// TwinCAT 3 PLC project TcLogTest
// ProgramVersion: 3.1.4023.0
// libraries:
//   Tc2_Standard, * (Beckhoff Automation GmbH)
//   Tc2_System, * (Beckhoff Automation GmbH)
//   Tc2_Utilities, * (Beckhoff Automation GmbH)
//   Tc3_Module, * (Beckhoff Automation GmbH)
//   TcLog, * (Benedikt Geisler)
//   TcUnit, * (www.tcunit.org)
// project tree:
//   / MAIN.TcPOU (not stored), PlcTask.TcTTO
//   TwinCAT/ ConvertAnyToString_TEST.TcPOU, DateTime_TEST.TcPOU, DynamicStringBuffer_TEST.TcPOU
//   NET/ TestWrapper_NET.TcPOU
// (motion and I/O tree: see PLC project tclog)
// real-time tasks:
//   TASK PlcTask1: cycle T#10ms, priority 21, ADS port 351

CONFIGURATION TcLogTest
    RESOURCE PLC ON TwinCAT3
        TASK PlcTask(INTERVAL := T#10ms, PRIORITY := 21);
        PROGRAM TESTS WITH PlcTask : TESTS;
    END_RESOURCE
END_CONFIGURATION

// ---- TwinCAT/ConvertAnyToString_TEST.TcPOU
FUNCTION_BLOCK ConvertAnyToString_TEST EXTENDS TcUnit.FB_TestSuite

ConvertAnyByteToString();
ConvertAnyDateAndTimeToString();
ConvertAnyDateToString();
ConvertAnyDINTToString();
ConvertAnyDTToString();
ConvertAnyINTToString();
ConvertAnyLINTToString();
ConvertAnyLRealToString();
ConvertAnyLWordToString();
ConvertAnyRealToString();
ConvertAnySINTToString();
ConvertAnyStringToString();
ConvertAnyTimeToString();
ConvertAnyTODToString();
ConvertAnyUDINTToString();
ConvertAnyUINTToString();
ConvertAnyULINTToString();
ConvertAnyUSINTToString();
ConvertAnyWordToString();
ConvertAnyWStringToString();

METHOD ConvertAnyByteToString : BOOL
VAR
	input : BYTE := 1;
	result : STRING;
	expected : STRING := '1';
END_VAR
TEST('ConvertAnyByteToString');
 
result := AnyToString(input);
 
AssertEquals(Expected := expected,
             Actual := result,
             Message := FormatResult(expected, result));
 
TEST_FINISHED();
END_METHOD

METHOD ConvertAnyDateAndTimeToString : BOOL
VAR
	input : DATE_AND_TIME := DT#1970-01-01-00:00;
	result : STRING;
	expected : STRING := 'DT#1970-01-01-00:00:00';
END_VAR
TEST('ConvertAnyDateAndTimeToString');
 
result := AnyToString(input);
 
AssertEquals(Expected := expected,
             Actual := result,
             Message := FormatResult(expected, result));
 
TEST_FINISHED();
END_METHOD

METHOD ConvertAnyDateToString : BOOL
VAR
	input : DATE := D#1970-01-01;
	result : STRING;
	expected : STRING := 'D#1970-01-01';
END_VAR
TEST('ConvertAnyDateToString');
 
result := AnyToString(input);
 
AssertEquals(Expected := expected,
             Actual := result,
             Message := FormatResult(expected, result));
 
TEST_FINISHED();
END_METHOD

METHOD ConvertAnyDINTToString : BOOL
VAR
	input : DINT := 1;
	result : STRING;
	expected : STRING := '1';
END_VAR
TEST('ConvertAnyDINTToString');
 
result := AnyToString(input);
 
AssertEquals(Expected := expected,
             Actual := result,
             Message := FormatResult(expected, result));
 
TEST_FINISHED();
END_METHOD

METHOD ConvertAnyDTToString : BOOL
VAR
	input : DT := DT#1970-01-01-00:00;
	result : STRING;
	expected : STRING := 'DT#1970-01-01-00:00:00';
END_VAR
TEST('ConvertAnyDTToString');
 
result := AnyToString(input);
 
AssertEquals(Expected := expected,
             Actual := result,
             Message := FormatResult(expected, result));
 
TEST_FINISHED();
END_METHOD

METHOD ConvertAnyDWordToString : BOOL
VAR
	input : DWORD := 1;
	result : STRING;
	expected : STRING := '1';
END_VAR
TEST('ConvertAnyDWordToString');
 
result := AnyToString(input);
 
AssertEquals(Expected := expected,
             Actual := result,
             Message := FormatResult(expected, result));
 
TEST_FINISHED();
END_METHOD

METHOD ConvertAnyINTToString : BOOL
VAR
	input : INT := 1;
	result : STRING;
	expected : STRING := '1';
END_VAR
TEST('ConvertAnyINTToString');
 
result := AnyToString(input);
 
AssertEquals(Expected := expected,
             Actual := result,
             Message := FormatResult(expected, result));
 
TEST_FINISHED();
END_METHOD

METHOD ConvertAnyLINTToString : BOOL
VAR
	input : LINT := 1;
	result : STRING;
	expected : STRING := '1';
END_VAR
TEST('ConvertAnyLINTToString');
 
result := AnyToString(input);
 
AssertEquals(Expected := expected,
             Actual := result,
             Message := FormatResult(expected, result));
 
TEST_FINISHED();
END_METHOD

METHOD ConvertAnyLRealToString : BOOL
VAR
	input : REAL := 1.0;
	result : STRING;
	expected : STRING := '1.0';
END_VAR
TEST('ConvertAnyRealToString');
 
result := AnyToString(input);
 
AssertEquals(Expected := expected,
             Actual := result,
             Message := FormatResult(expected, result));
 
TEST_FINISHED();
END_METHOD

METHOD ConvertAnyLWordToString : BOOL
VAR
	input : LWORD := 1;
	result : STRING;
	expected : STRING := '1';
END_VAR
TEST('ConvertAnyLWordToString');
 
result := AnyToString(input);
 
AssertEquals(Expected := expected,
             Actual := result,
             Message := FormatResult(expected, result));
 
TEST_FINISHED();
END_METHOD

METHOD ConvertAnyRealToString : BOOL
VAR
	input : LREAL := 1.0;
	result : STRING;
	expected : STRING := '1.0';
END_VAR
TEST('ConvertAnyLRealToString');
 
result := AnyToString(input);
 
AssertEquals(Expected := expected,
             Actual := result,
             Message := FormatResult(expected, result));
 
TEST_FINISHED();
END_METHOD

METHOD ConvertAnySINTToString : BOOL
VAR
	input : SINT := 1;
	result : STRING;
	expected : STRING := '1';
END_VAR
TEST('ConvertAnySINTToString');
 
result := AnyToString(input);
 
AssertEquals(Expected := expected,
             Actual := result,
             Message := FormatResult(expected, result));
 
TEST_FINISHED();
END_METHOD

METHOD ConvertAnyStringToString : BOOL
VAR
	input : STRING := 'Hallo';
	result : STRING;
	expected : STRING := 'Hallo';
END_VAR
TEST('ConvertAnyStringToString');
 
result := AnyToString(input);
 
AssertEquals(Expected := expected,
             Actual := result,
             Message := FormatResult(expected, result));
 
TEST_FINISHED();
END_METHOD

METHOD ConvertAnyTimeToString : BOOL
VAR
	input : TIME := T#49D17H2M47S295MS;
	result : STRING;
	expected : STRING := 'T#49d17h2m47s295ms';
END_VAR
TEST('ConvertAnyTimeToString');
 
result := AnyToString(input);
 
AssertEquals(Expected := expected,
             Actual := result,
             Message := FormatResult(expected, result));
 
TEST_FINISHED();
END_METHOD

METHOD ConvertAnyTODToString : BOOL
VAR
	input : TOD := TOD#11:02:47.295;
	result : STRING;
	expected : STRING := 'TOD#11:02:47.295';
END_VAR
TEST('ConvertAnyTODToString');
 
result := AnyToString(input);
 
AssertEquals(Expected := expected,
             Actual := result,
             Message := FormatResult(expected, result));
 
TEST_FINISHED();
END_METHOD

METHOD ConvertAnyUDINTToString : BOOL
VAR
	input : UDINT := 1;
	result : STRING;
	expected : STRING := '1';
END_VAR
TEST('ConvertAnyUDINTToString');
 
result := AnyToString(input);
 
AssertEquals(Expected := expected,
             Actual := result,
             Message := FormatResult(expected, result));
 
TEST_FINISHED();
END_METHOD

METHOD ConvertAnyUINTToString : BOOL
VAR
	input : UINT := 1;
	result : STRING;
	expected : STRING := '1';
END_VAR
TEST('ConvertAnyUINTToString');
 
result := AnyToString(input);
 
AssertEquals(Expected := expected,
             Actual := result,
             Message := FormatResult(expected, result));
 
TEST_FINISHED();
END_METHOD

METHOD ConvertAnyULINTToString : BOOL
VAR
	input : ULINT := 1;
	result : STRING;
	expected : STRING := '1';
END_VAR
TEST('ConvertAnyULINTToString');
 
result := AnyToString(input);
 
AssertEquals(Expected := expected,
             Actual := result,
             Message := FormatResult(expected, result));
 
TEST_FINISHED();
END_METHOD

METHOD ConvertAnyUSINTToString : BOOL
VAR
	input : USINT := 1;
	result : STRING;
	expected : STRING := '1';
END_VAR
TEST('ConvertAnyUSINTToString');
 
result := AnyToString(input);
 
AssertEquals(Expected := expected,
             Actual := result,
             Message := FormatResult(expected, result));
 
TEST_FINISHED();
END_METHOD

METHOD ConvertAnyWordToString : BOOL
VAR
	input : WORD := 1;
	result : STRING;
	expected : STRING := '1';
END_VAR
TEST('ConvertAnyWordToString');
 
result := AnyToString(input);
 
AssertEquals(Expected := expected,
             Actual := result,
             Message := FormatResult(expected, result));
 
TEST_FINISHED();
END_METHOD

METHOD ConvertAnyWStringToString : BOOL
VAR
	input : WSTRING := "Hallo";
	result : STRING;
	expected : STRING := 'Hallo';
END_VAR
TEST('ConvertAnyWStringToString');
 
result := AnyToString(input);
 
AssertEquals(Expected := expected,
             Actual := result,
             Message := FormatResult(expected, result));
 
TEST_FINISHED();
END_METHOD

METHOD PRIVATE FormatResult : STRING
VAR_INPUT
	Expected : STRING;
	Result : STRING;
END_VAR
FormatResult := Tc2_Standard.CONCAT('Conversion failed. Expected: ', Tc2_Standard.CONCAT(Expected, Tc2_Standard.CONCAT(' - Result: ', Result)));
END_METHOD

END_FUNCTION_BLOCK

// ---- TwinCAT/DateTime_TEST.TcPOU
FUNCTION_BLOCK DateTime_TEST EXTENDS TcUnit.FB_TestSuite

CheckStringFormat();

METHOD CheckStringFormat
VAR_INST
	sut : DateTime;
	expected : STRING;
	result : STRING;
END_VAR
VAR
	localSystemTime : Tc2_Utilities.TIMESTRUCT;
END_VAR
sut();

TEST('CheckStringFormat');

localSystemTime := sut.AsLocalSystemTime;

expected := Tc2_Standard.CONCAT('-', TO_STRING(localSystemTime.wYear));
IF localSystemTime.wMonth < 10 THEN expected := Tc2_Standard.CONCAT(expected, '0'); END_IF
expected := Tc2_Standard.CONCAT(expected, TO_STRING(localSystemTime.wMonth));
IF localSystemTime.wDay < 10 THEN expected := Tc2_Standard.CONCAT(expected, '0'); END_IF
expected := Tc2_Standard.CONCAT(expected, TO_STRING(localSystemTime.wDay));
expected := Tc2_Standard.CONCAT(expected, '-');
IF localSystemTime.wHour < 10 THEN expected := Tc2_Standard.CONCAT(expected, '0'); END_IF
expected := Tc2_Standard.CONCAT(expected, TO_STRING(localSystemTime.wHour));
expected := Tc2_Standard.CONCAT(expected, ':');
IF localSystemTime.wMinute < 10 THEN expected := Tc2_Standard.CONCAT(expected, '0'); END_IF
expected := Tc2_Standard.CONCAT(expected, TO_STRING(localSystemTime.wMinute));
expected := Tc2_Standard.CONCAT(expected, ':');
IF localSystemTime.wSecond < 10 THEN expected := Tc2_Standard.CONCAT(expected, '0'); END_IF
expected := Tc2_Standard.CONCAT(expected, TO_STRING(localSystemTime.wSecond));
expected := Tc2_Standard.CONCAT(expected, '-');

result := sut.ToFormatString('-YYYYMMDD-hh:mm:ss-');
	
IF sut.Done THEN
	AssertEquals(
		Expected 	:= 	expected,
		Actual 		:=  result,
		Message		:=	'Time formatting failed.'
	);

	TEST_FINISHED();
END_IF
END_METHOD

END_FUNCTION_BLOCK

// ---- TwinCAT/DynamicStringBuffer_TEST.TcPOU
FUNCTION_BLOCK DynamicStringBuffer_TEST EXTENDS FB_TestSuite

LogsManyMessagesForManyCycles();

METHOD LogsManyMessagesForManyCycles
VAR
	result : STRING := '';
	expected : STRING := '';
	i : UDINT;
END_VAR
VAR CONSTANT
	Cycles : UDINT := 50;
	Messages : UDINT := 50;
END_VAR
VAR_INST
	cycleCount : UDINT := 0;
	logsManyMessagesForManyCyclesLogger : TcLogCore(BufferSize:=50 * 50 * 280); // Cycles * Messages * (max string length + fifo overhead (estimated))
	logger : TcLog;
END_VAR
TEST('LogsManyMessagesForManyCycles');

logsManyMessagesForManyCyclesLogger
	.WriteToFile('c:\UnitTest\', 'test.txt')
	.RunLogger();
logger.SetLogger(logsManyMessagesForManyCyclesLogger);

IF cycleCount < Cycles THEN
	FOR i:=0 TO Messages DO
		logger
			.AppendString('Cycle: ')
			.AppendString(UDINT_TO_STRING(cycleCount))
			.AppendString(', Message: ')
			.AppendString(UDINT_TO_STRING(i))
			.Error('');	
	END_FOR
END_IF
cycleCount := cycleCount + 1;

// Catch any occuring error message
IF LEN(logsManyMessagesForManyCyclesLogger.Error.Info) > 0 THEN
	result := logsManyMessagesForManyCyclesLogger.Error.Info;
END_IF

IF cycleCount > (Cycles * Messages * 2 + 4) THEN 
	AssertEquals(Expected := expected,
				 Actual := result,
				 Message := result);
 
	TEST_FINISHED();
END_IF
END_METHOD

END_FUNCTION_BLOCK

// ---- NET/TestWrapper_NET.TcPOU
FUNCTION_BLOCK TestWrapper_NET
VAR
	_coreLogger : TcLogCore(BufferSize:=50 * 50 * 280);
	_logger : TcLog;
	_flushCache : BOOL;
	
	// Test drivers
	_getDateTime : DateTime;
	_setLocalSystemTime : NT_SetLocalTime;
	_cycles : INT;
	_i : INT;
	_persistenceTimeStaysWithinBounds : F_TRIG;
	
	// Exchanged variables with .NET tests
	FilePath : STRING;
	FileName : STRING;
	Delimiter : STRING(1);
	NewLocalSystemTimeToBeSet : STRING;
	TriggerNewLocalSystemTime : BOOL;
	LocalTimeAsString : STRING;
	
	Persist_simple_error_message_run : BOOL;
	Persist_simple_error_message_data : STRING;
	
	Persist_long_error_message_run : BOOL;
	Persist_long_error_message_data : T_MaxString;
	
	Do_not_persist_logs_below_log_level_run : BOOL;
	
	Log_message_contains_instance_path_run : BOOL;
	
	Log_message_uses_correct_delimiter_run : BOOL;
	Log_message_uses_correct_delimiter_data : STRING;
	
	Log_message_contains_custom_formatted_timestamp_run : BOOL;
	
	Delete_logs_if_expired_run : BOOL;
	
	New_logfile_is_created_if_rolling_interval_rolls_run : BOOL;
	
	Same_log_file_is_used_until_rolling_interval_rolls : BOOL;
	
	Log_in_consecutive_cycles : BOOL;
	Number_of_log_cycles : DINT;
	
	Log_multiple_logs_in_one_cycle : BOOL;
	Number_of_logs_per_cycle : DINT;
	
	Log_multiple_logs_in_multiple_cycles : BOOL;
	Number_of_cycles : DINT;
	CycleCount : DINT := 1;
	
	Persistance_time_stays_within_bounds : BOOL;
	Duration_in_cylces : DINT := 1;
END_VAR

// ****** U N I T   T E S T S ******

// Set up TcLog
_coreLogger
	.IncludeInstancePath()
	.MinimumLevel(LogLevels.Warning)
	.SetDelimiter(Delimiter)
	.SetRollingInterval(RollingIntervals.Hourly)
	.DeleteLogFilesAfterDays(1)
	.TimestampFormat('_YYMMDD-hh-mm-ss_')
	.WriteToAds()
	.WriteToFile(FilePath, FileName)
	.RunLogger();

IF _flushCache THEN _coreLogger.FlushCache(); END_IF
	
// Test drivers
_getDateTime();
LocalTimeAsString := _getDateTime.AsLocalSystemTimeString;

_setLocalSystemTime(
	NETID 	:= '',
	TIMESTR := STRING_TO_SYSTEMTIME(NewLocalSystemTimeToBeSet),
	START 	:= TriggerNewLocalSystemTime,
	TMOUT	:= T#2S
	);

// Execute tests
IF Persist_simple_error_message_run THEN
	Persist_simple_error_message_run := FALSE;
	_logger
		.Error(Persist_simple_error_message_data);
END_IF

IF Persist_long_error_message_run THEN
	Persist_long_error_message_run := FALSE;
	_logger
		.Error(Persist_long_error_message_data);
END_IF

IF Do_not_persist_logs_below_log_level_run THEN
	Do_not_persist_logs_below_log_level_run := FALSE;
	_logger
		.Information('Nothing');
END_IF

IF Log_message_contains_instance_path_run THEN
	Log_message_contains_instance_path_run := FALSE;
	_logger
		.Error('Nothing');
END_IF

IF Log_message_uses_correct_delimiter_run THEN
	Log_message_uses_correct_delimiter_run := FALSE;
	_logger
		.Error(Log_message_uses_correct_delimiter_data);
END_IF

IF Log_message_contains_custom_formatted_timestamp_run THEN
	Log_message_contains_custom_formatted_timestamp_run := FALSE;
	_logger
		.Error('Test message');
END_IF

IF Delete_logs_if_expired_run THEN
	Delete_logs_if_expired_run := FALSE;
	_logger
		.Error('Test message');
END_IF

IF New_logfile_is_created_if_rolling_interval_rolls_run THEN
	New_logfile_is_created_if_rolling_interval_rolls_run := FALSE;
	_logger
		.Error('Test message');
END_IF

IF Same_log_file_is_used_until_rolling_interval_rolls THEN
	Same_log_file_is_used_until_rolling_interval_rolls := FALSE;
	_logger
		.Error('Test message');
END_IF

IF Log_in_consecutive_cycles THEN
	_logger
		.Error(Tc2_Standard.CONCAT('Logging cycle ', INT_TO_STRING(_cycles)));
	_cycles := _cycles + 1;
	IF _cycles >= Number_of_log_cycles THEN
		_cycles := 0;
		Log_in_consecutive_cycles := FALSE;
	END_IF
END_IF

IF Log_multiple_logs_in_one_cycle THEN
	FOR _i:= 1 TO DINT_TO_INT(Number_of_logs_per_cycle) DO
		_logger.
			Error(Tc2_Standard.CONCAT('Logging multiple times per cycle. Current step: ', INT_TO_STRING(_i))); 
	END_FOR
	Log_multiple_logs_in_one_cycle := FALSE;
END_IF

IF Log_multiple_logs_in_multiple_cycles THEN
	IF CycleCount <= Number_of_cycles THEN	
		FOR _i:= 1 TO DINT_TO_INT(Number_of_logs_per_cycle) DO
			_logger
				.AppendString('Logging multiple times per cycle. Cycle: ')
				.AppendString(DINT_TO_STRING(CycleCount))
				.AppendString(' / Step: ')
				.AppendString(INT_TO_STRING(_i))
				.Error('');
		END_FOR
		CycleCount := CycleCount + 1;
	ELSE
		CycleCount := 1;
		Log_multiple_logs_in_multiple_cycles := FALSE;
	END_IF
END_IF 

_persistenceTimeStaysWithinBounds(CLK := (Persistance_time_stays_within_bounds AND _coreLogger.Busy));
IF _persistenceTimeStaysWithinBounds.Q THEN
	CycleCount := 1;
	Persistance_time_stays_within_bounds := FALSE;
END_IF
IF Persistance_time_stays_within_bounds THEN
	Duration_in_cylces := Duration_in_cylces + 1;
	IF CycleCount <= Number_of_cycles THEN	
		FOR _i:= 1 TO DINT_TO_INT(Number_of_logs_per_cycle) DO
			_logger
				.AppendString('Logging multiple times per cycle. Cycle: ')
				.AppendString(DINT_TO_STRING(CycleCount))
				.AppendString(' / Step: ')
				.AppendString(INT_TO_STRING(_i))
				.Error('');
		END_FOR
		CycleCount := CycleCount + 1;
	END_IF
END_IF

END_FUNCTION_BLOCK
